(* IEC 61131-3 sources: NVM-AquaFeed-Platform/02_Software_Design/PLC/07_Implementation/Function_Blocks (part 2) *)

(* ---- FB_LineManager.st ---- *)
FUNCTION_BLOCK FB_LineManager
VAR_INPUT
    xEnableFromSystem : BOOL;
    xStart : BOOL;
    xPause : BOOL;
    xStop : BOOL;
    xCancel : BOOL;
    udiCommandSequence : UDINT;
    udiResetSequence : UDINT;
    xEmergencyStop : BOOL;
    xSafetyOK : BOOL;
    xBlockingFault : BOOL;
    xDesktopCommunicationOK : BOOL;
    stConfig : ST_LineConfig;
    udiMonotonicTickMs : UDINT;

    xJobAvailable : BOOL;
    xAcceptJob : BOOL;
    xCandidateIntegrityValid : BOOL;
    stJobCandidate : ST_JobExecution;
    stRecipeCandidate : ST_RecipeExecution;

    xSelectorReady : BOOL;
    xSelectorInPosition : BOOL;
    uiSelectorOutlet : UINT;
    xSelectorFault : BOOL;

    xBlowerReady : BOOL;
    xBlowerRunning : BOOL;
    xBlowerAtSpeed : BOOL;
    xBlowerDosingPermitted : BOOL;
    xBlowerFault : BOOL;

    xDosing1Ready : BOOL;
    xDosing1Running : BOOL;
    xDosing1Fault : BOOL;
    xDosing1CompletedEvent : BOOL;
    udiDosing1DeliveredCentiKg : UDINT;
    udiDosing1IncrementCentiKg : UDINT;

    xDosing2Ready : BOOL;
    xDosing2Running : BOOL;
    xDosing2Fault : BOOL;
    xDosing2CompletedEvent : BOOL;
    udiDosing2DeliveredCentiKg : UDINT;
    udiDosing2IncrementCentiKg : UDINT;
END_VAR
VAR_OUTPUT
    stLine : ST_Line;
    xReady : BOOL;
    xBusy : BOOL;
    xCompleted : BOOL;
    xJobAccepted : BOOL;
    xJobRejected : BOOL;
    uiResultCode : UINT;
    udiLastAcceptedCommandSequence : UDINT;

    xSelectorMoveRequest : BOOL;
    uiSelectorTargetOutlet : UINT;
    udiSelectorCommandSequence : UDINT;

    xBlowerRunRequest : BOOL;
    xBlowerNormalStopRequest : BOOL;
    uiBlowerTargetFreqCentiHz : UINT;
    udiBlowerRequestedPostRunTimeMs : UDINT;
    udiBlowerCommandSequence : UDINT;

    xDosing1StartRequest : BOOL;
    xDosing1StopRequest : BOOL;
    udiDosing1CommandSequence : UDINT;
    udiDosing1JobId : UDINT;
    uiDosing1OutletId : UINT;
    udiDosing1TargetCentiKg : UDINT;
    uiDosing1SpeedPermille : UINT;

    xDosing2StartRequest : BOOL;
    xDosing2StopRequest : BOOL;
    udiDosing2CommandSequence : UDINT;
    udiDosing2JobId : UDINT;
    uiDosing2OutletId : UINT;
    udiDosing2TargetCentiKg : UDINT;
    uiDosing2SpeedPermille : UINT;

    xEquipmentResetRequest : BOOL;
    udiEquipmentResetSequence : UDINT;
END_VAR
VAR
    eState : E_LineState := LINE_OFF;
    stAcceptedJob : ST_JobExecution;
    stAcceptedRecipe : ST_RecipeExecution;
    xActiveJobValid : BOOL;
    xConfigValid : BOOL;
    xCandidateValid : BOOL;
    xSelectedDosingReady : BOOL;
    xSelectedDosingRunning : BOOL;
    xSelectedDosingFault : BOOL;
    xSelectedDosingComplete : BOOL;
    udiSelectedDosingIncrement : UDINT;
    udiSelectedDosingTarget : UDINT;
    udiExecutionStartTickMs : UDINT;
    udiStateStartTickMs : UDINT;
    udiLastResetSequence : UDINT;
    udiLastProcessedTransferSequence : UDINT;
    udiInternalCommandSequence : UDINT;
    xHasAcceptedCommand : BOOL;
    xHasAcceptedReset : BOOL;
    xHasProcessedTransfer : BOOL;
    xShutdownForPause : BOOL;
    xShutdownForCancel : BOOL;
    xShutdownForStop : BOOL;
    xSelectorSettleTimerActive : BOOL;
    xCompleteEventIssued : BOOL;
END_VAR
VAR CONSTANT
    c_udiMaximumProgressTarget : UDINT := 4000000;
    c_udiMaximumExecutionTimeSec : UDINT := 4294967;
    c_uiResultNone : UINT := 0;
    c_uiResultAccepted : UINT := 1;
    c_uiResultCompleted : UINT := 2;
    c_uiResultStopped : UINT := 3;
    c_uiResultCancelled : UINT := 4;
    c_uiResultInvalidConfig : UINT := 60;
    c_uiResultDesktopOffline : UINT := 61;
    c_uiResultIntegrity : UINT := 62;
    c_uiResultInvalidCandidate : UINT := 63;
    c_uiResultEquipmentNotReady : UINT := 64;
    c_uiResultEquipmentFault : UINT := 65;
    c_uiResultSafety : UINT := 66;
    c_uiResultEmergency : UINT := 67;
    c_uiResultTimeout : UINT := 68;
    c_uiResultSequenceOverflow : UINT := 69;
    c_uiResultArithmetic : UINT := 70;
END_VAR

xReady := FALSE;
xBusy := xActiveJobValid;
xCompleted := FALSE;
xJobAccepted := FALSE;
xJobRejected := FALSE;
xSelectorMoveRequest := FALSE;
uiSelectorTargetOutlet := 0;
xBlowerRunRequest := FALSE;
xBlowerNormalStopRequest := FALSE;
uiBlowerTargetFreqCentiHz := 0;
udiBlowerRequestedPostRunTimeMs := 0;
xDosing1StartRequest := FALSE;
xDosing1StopRequest := FALSE;
udiDosing1JobId := 0;
uiDosing1OutletId := 0;
udiDosing1TargetCentiKg := 0;
uiDosing1SpeedPermille := 0;
xDosing2StartRequest := FALSE;
xDosing2StopRequest := FALSE;
udiDosing2JobId := 0;
uiDosing2OutletId := 0;
udiDosing2TargetCentiKg := 0;
uiDosing2SpeedPermille := 0;
xEquipmentResetRequest := FALSE;

xConfigValid := (stConfig.usiLineId > 0) AND
                (stConfig.uiSelectorOutletCount > 0) AND
                (stConfig.uiSelectorOutletCount <= 64) AND
                (stConfig.xDosing1Enabled OR
                 stConfig.xDosing2Enabled) AND
                (stConfig.udiMaximumTargetCentiKg > 0) AND
                (stConfig.udiMaximumTargetCentiKg <=
                 c_udiMaximumProgressTarget) AND
                (stConfig.udiMaximumFeedToleranceCentiKg <
                 stConfig.udiMaximumTargetCentiKg) AND
                (stConfig.uiMinimumDosingSpeedPermille > 0) AND
                (stConfig.uiMinimumDosingSpeedPermille <=
                 stConfig.uiMaximumDosingSpeedPermille) AND
                (stConfig.uiMaximumDosingSpeedPermille <= 1000) AND
                (stConfig.uiMinimumBlowerFreqCentiHz > 0) AND
                (stConfig.uiMinimumBlowerFreqCentiHz <=
                 stConfig.uiMaximumBlowerFreqCentiHz) AND
                (stConfig.udiMaximumSelectorSettleTimeMs > 0) AND
                (stConfig.udiMaximumBlowerPreRunTimeMs > 0) AND
                (stConfig.udiMaximumBlowerPostRunTimeMs > 0) AND
                (stConfig.udiMaximumDosingTimeSec > 0) AND
                (stConfig.udiMaximumExecutionTimeSec > 0) AND
                (stConfig.udiMaximumExecutionTimeSec <=
                 c_udiMaximumExecutionTimeSec);

xCandidateValid := xJobAvailable AND
                   xCandidateIntegrityValid AND
                   (stJobCandidate.uiSnapshotVersion = 1) AND
                   (stRecipeCandidate.uiSnapshotVersion = 1) AND
                   (stJobCandidate.udiJobId > 0) AND
                   (stJobCandidate.usiLineId =
                    stConfig.usiLineId) AND
                   (stJobCandidate.uiRecipeId > 0) AND
                   (stJobCandidate.uiRecipeId =
                    stRecipeCandidate.uiRecipeId) AND
                   (stJobCandidate.udiRecipeRevision =
                    stRecipeCandidate.udiRecipeRevision) AND
                   (stJobCandidate.uiTargetSelectorOutlet > 0) AND
                   (stJobCandidate.uiTargetSelectorOutlet <=
                    stConfig.uiSelectorOutletCount) AND
                   (((stJobCandidate.byDosingUnitMask = 16#01) AND
                     stConfig.xDosing1Enabled) OR
                    ((stJobCandidate.byDosingUnitMask = 16#02) AND
                     stConfig.xDosing2Enabled)) AND
                   (stJobCandidate.udiTargetFeedCentiKg > 0) AND
                   (stJobCandidate.udiTargetFeedCentiKg <=
                    stConfig.udiMaximumTargetCentiKg) AND
                   (stRecipeCandidate.udiFeedToleranceCentiKg <=
                    stConfig.udiMaximumFeedToleranceCentiKg) AND
                   (stRecipeCandidate.udiFeedToleranceCentiKg <
                    stJobCandidate.udiTargetFeedCentiKg) AND
                   (stRecipeCandidate.uiDosingSpeedPermille >=
                    stConfig.uiMinimumDosingSpeedPermille) AND
                   (stRecipeCandidate.uiDosingSpeedPermille <=
                    stConfig.uiMaximumDosingSpeedPermille) AND
                   (stRecipeCandidate.uiBlowerFreqCentiHz >=
                    stConfig.uiMinimumBlowerFreqCentiHz) AND
                   (stRecipeCandidate.uiBlowerFreqCentiHz <=
                    stConfig.uiMaximumBlowerFreqCentiHz) AND
                   (stRecipeCandidate.udiSelectorSettleTimeMs <=
                    stConfig.udiMaximumSelectorSettleTimeMs) AND
                   (stRecipeCandidate.udiBlowerPreRunTimeMs <=
                    stConfig.udiMaximumBlowerPreRunTimeMs) AND
                   (stRecipeCandidate.udiBlowerPostRunTimeMs > 0) AND
                   (stRecipeCandidate.udiBlowerPostRunTimeMs <=
                    stConfig.udiMaximumBlowerPostRunTimeMs) AND
                   (stRecipeCandidate.udiMaximumDosingTimeSec > 0) AND
                   (stRecipeCandidate.udiMaximumDosingTimeSec <=
                    stConfig.udiMaximumDosingTimeSec) AND
                   (stJobCandidate.udiMaximumExecutionTimeSec > 0) AND
                   (stJobCandidate.udiMaximumExecutionTimeSec <=
                    stConfig.udiMaximumExecutionTimeSec);

xSelectedDosingReady := FALSE;
xSelectedDosingRunning := FALSE;
xSelectedDosingFault := FALSE;
xSelectedDosingComplete := FALSE;
udiSelectedDosingIncrement := 0;

IF xActiveJobValid THEN
    IF stAcceptedJob.byDosingUnitMask = 16#01 THEN
        xSelectedDosingReady := xDosing1Ready;
        xSelectedDosingRunning := xDosing1Running;
        xSelectedDosingFault := xDosing1Fault;
        xSelectedDosingComplete := xDosing1CompletedEvent;
        udiSelectedDosingIncrement :=
            udiDosing1IncrementCentiKg;
    ELSIF stAcceptedJob.byDosingUnitMask = 16#02 THEN
        xSelectedDosingReady := xDosing2Ready;
        xSelectedDosingRunning := xDosing2Running;
        xSelectedDosingFault := xDosing2Fault;
        xSelectedDosingComplete := xDosing2CompletedEvent;
        udiSelectedDosingIncrement :=
            udiDosing2IncrementCentiKg;
    END_IF;
END_IF;

IF NOT xEnableFromSystem THEN
    eState := LINE_OFF;
    xActiveJobValid := FALSE;
    xShutdownForPause := FALSE;
    xShutdownForCancel := FALSE;
    xShutdownForStop := FALSE;
    xCompleteEventIssued := FALSE;
    uiResultCode := c_uiResultNone;
ELSIF NOT xConfigValid THEN
    eState := LINE_FAULT;
    uiResultCode := c_uiResultInvalidConfig;
ELSIF xEmergencyStop THEN
    eState := LINE_EMERGENCY;
    uiResultCode := c_uiResultEmergency;
ELSIF xActiveJobValid AND
      (NOT xSafetyOK OR xBlockingFault) THEN
    eState := LINE_FAULT;
    uiResultCode := c_uiResultSafety;
ELSIF xActiveJobValid AND
      (xSelectorFault OR xBlowerFault OR
       xSelectedDosingFault) THEN
    eState := LINE_FAULT;
    uiResultCode := c_uiResultEquipmentFault;
ELSE
    IF xActiveJobValid AND
       (eState <> LINE_PAUSED) AND
       (eState <> LINE_FAULT) AND
       (eState <> LINE_EMERGENCY) AND
       (F_ElapsedMs(udiCurrentTickMs := udiMonotonicTickMs,
                    udiStartTickMs := udiExecutionStartTickMs) >=
        (stAcceptedJob.udiMaximumExecutionTimeSec * 1000)) THEN
        eState := LINE_FAULT;
        uiResultCode := c_uiResultTimeout;
    END_IF;

    IF xActiveJobValid AND
       (eState <> LINE_LOAD_JOB) AND
       (eState <> LINE_READY) AND
       (eState <> LINE_PAUSED) AND
       (eState <> LINE_FAULT) AND
       (eState <> LINE_EMERGENCY) AND
       (NOT xHasAcceptedCommand OR
        (udiCommandSequence <>
         udiLastAcceptedCommandSequence)) THEN
        IF xCancel OR xStop OR xPause THEN
            udiLastAcceptedCommandSequence :=
                udiCommandSequence;
            xHasAcceptedCommand := TRUE;
            xShutdownForCancel := xCancel;
            xShutdownForStop := xStop AND NOT xCancel;
            xShutdownForPause :=
                xPause AND NOT xStop AND NOT xCancel;
            eState := LINE_STOP_DOSING;
        END_IF;
    END_IF;

    CASE eState OF
        LINE_OFF:
            eState := LINE_INITIALIZING;
            uiResultCode := c_uiResultNone;

        LINE_INITIALIZING:
            IF xSafetyOK AND
               NOT xBlockingFault AND
               NOT xSelectorFault AND
               NOT xBlowerFault THEN
                eState := LINE_READY;
            END_IF;

        LINE_READY:
            xReady := TRUE;

            IF xAcceptJob AND
               (NOT xHasProcessedTransfer OR
                (stJobCandidate.udiTransferSequence <>
                 udiLastProcessedTransferSequence)) THEN
                udiLastProcessedTransferSequence :=
                    stJobCandidate.udiTransferSequence;
                xHasProcessedTransfer := TRUE;

                IF NOT xDesktopCommunicationOK THEN
                    xJobRejected := TRUE;
                    uiResultCode := c_uiResultDesktopOffline;
                ELSIF NOT xCandidateIntegrityValid THEN
                    xJobRejected := TRUE;
                    uiResultCode := c_uiResultIntegrity;
                ELSIF NOT xCandidateValid THEN
                    xJobRejected := TRUE;
                    uiResultCode := c_uiResultInvalidCandidate;
                ELSE
                    stAcceptedJob := stJobCandidate;
                    stAcceptedRecipe := stRecipeCandidate;
                    xActiveJobValid := TRUE;
                    xJobAccepted := TRUE;
                    xShutdownForPause := FALSE;
                    xShutdownForCancel := FALSE;
                    xShutdownForStop := FALSE;
                    xCompleteEventIssued := FALSE;
                    stLine.udiDeliveredFeedCentiKg := 0;
                    uiResultCode := c_uiResultAccepted;
                    eState := LINE_LOAD_JOB;
                END_IF;
            END_IF;

        LINE_LOAD_JOB:
            IF xStart AND
               (NOT xHasAcceptedCommand OR
                (udiCommandSequence <>
                 udiLastAcceptedCommandSequence)) THEN
                udiLastAcceptedCommandSequence :=
                    udiCommandSequence;
                xHasAcceptedCommand := TRUE;
                udiExecutionStartTickMs :=
                    udiMonotonicTickMs;
                eState := LINE_VALIDATE;
            END_IF;

        LINE_VALIDATE:
            IF NOT xSafetyOK OR xBlockingFault OR
               NOT xSelectorReady OR
               NOT xBlowerReady OR
               NOT xSelectedDosingReady THEN
                eState := LINE_FAULT;
                uiResultCode := c_uiResultEquipmentNotReady;
            ELSIF udiInternalCommandSequence =
                  16#FFFFFFFF THEN
                eState := LINE_FAULT;
                uiResultCode := c_uiResultSequenceOverflow;
            ELSE
                udiInternalCommandSequence :=
                    udiInternalCommandSequence + 1;
                udiSelectorCommandSequence :=
                    udiInternalCommandSequence;
                eState := LINE_MOVE_SELECTOR;
            END_IF;

        LINE_MOVE_SELECTOR:
            xSelectorMoveRequest := TRUE;
            uiSelectorTargetOutlet :=
                stAcceptedJob.uiTargetSelectorOutlet;
            eState := LINE_WAIT_SELECTOR;
            xSelectorSettleTimerActive := FALSE;

        LINE_WAIT_SELECTOR:
            uiSelectorTargetOutlet :=
                stAcceptedJob.uiTargetSelectorOutlet;

            IF xSelectorInPosition AND
               (uiSelectorOutlet =
                stAcceptedJob.uiTargetSelectorOutlet) THEN
                IF NOT xSelectorSettleTimerActive THEN
                    udiStateStartTickMs :=
                        udiMonotonicTickMs;
                    xSelectorSettleTimerActive := TRUE;
                ELSIF F_ElapsedMs(
                          udiCurrentTickMs :=
                              udiMonotonicTickMs,
                          udiStartTickMs :=
                              udiStateStartTickMs) >=
                      stAcceptedRecipe.
                          udiSelectorSettleTimeMs THEN
                    eState := LINE_START_BLOWER;
                END_IF;
            ELSE
                xSelectorSettleTimerActive := FALSE;
            END_IF;

        LINE_START_BLOWER:
            IF udiInternalCommandSequence =
               16#FFFFFFFF THEN
                eState := LINE_FAULT;
                uiResultCode := c_uiResultSequenceOverflow;
            ELSE
                udiInternalCommandSequence :=
                    udiInternalCommandSequence + 1;
                udiBlowerCommandSequence :=
                    udiInternalCommandSequence;
                eState := LINE_WAIT_BLOWER;
            END_IF;

        LINE_WAIT_BLOWER:
            xBlowerRunRequest := TRUE;
            uiBlowerTargetFreqCentiHz :=
                stAcceptedRecipe.uiBlowerFreqCentiHz;
            udiBlowerRequestedPostRunTimeMs :=
                stAcceptedRecipe.udiBlowerPostRunTimeMs;

            IF xBlowerAtSpeed AND
               xBlowerDosingPermitted THEN
                udiStateStartTickMs :=
                    udiMonotonicTickMs;
                eState := LINE_PRE_RUN;
            END_IF;

        LINE_PRE_RUN:
            xBlowerRunRequest := TRUE;
            uiBlowerTargetFreqCentiHz :=
                stAcceptedRecipe.uiBlowerFreqCentiHz;
            udiBlowerRequestedPostRunTimeMs :=
                stAcceptedRecipe.udiBlowerPostRunTimeMs;

            IF NOT xSelectorInPosition OR
               (uiSelectorOutlet <>
                stAcceptedJob.uiTargetSelectorOutlet) OR
               NOT xBlowerDosingPermitted THEN
                eState := LINE_FAULT;
                uiResultCode := c_uiResultEquipmentFault;
            ELSIF F_ElapsedMs(
                      udiCurrentTickMs :=
                          udiMonotonicTickMs,
                      udiStartTickMs :=
                          udiStateStartTickMs) >=
                  stAcceptedRecipe.
                      udiBlowerPreRunTimeMs THEN
                eState := LINE_START_DOSING;
            END_IF;

        LINE_START_DOSING:
            xBlowerRunRequest := TRUE;
            uiBlowerTargetFreqCentiHz :=
                stAcceptedRecipe.uiBlowerFreqCentiHz;
            udiBlowerRequestedPostRunTimeMs :=
                stAcceptedRecipe.udiBlowerPostRunTimeMs;

            IF udiInternalCommandSequence =
               16#FFFFFFFF THEN
                eState := LINE_FAULT;
                uiResultCode := c_uiResultSequenceOverflow;
            ELSE
                udiInternalCommandSequence :=
                    udiInternalCommandSequence + 1;
                IF stAcceptedJob.byDosingUnitMask =
                   16#01 THEN
                    udiDosing1CommandSequence :=
                        udiInternalCommandSequence;
                ELSE
                    udiDosing2CommandSequence :=
                        udiInternalCommandSequence;
                END_IF;

                IF stLine.udiDeliveredFeedCentiKg >=
                   stAcceptedJob.udiTargetFeedCentiKg THEN
                    udiSelectedDosingTarget := 0;
                ELSE
                    udiSelectedDosingTarget :=
                        stAcceptedJob.
                            udiTargetFeedCentiKg -
                        stLine.
                            udiDeliveredFeedCentiKg;
                END_IF;
                eState := LINE_FEEDING;
            END_IF;

        LINE_FEEDING:
            xBlowerRunRequest := TRUE;
            uiBlowerTargetFreqCentiHz :=
                stAcceptedRecipe.uiBlowerFreqCentiHz;
            udiBlowerRequestedPostRunTimeMs :=
                stAcceptedRecipe.udiBlowerPostRunTimeMs;

            IF stAcceptedJob.byDosingUnitMask = 16#01 THEN
                xDosing1StartRequest := TRUE;
                udiDosing1JobId := stAcceptedJob.udiJobId;
                uiDosing1OutletId :=
                    stAcceptedJob.uiTargetSelectorOutlet;
                udiDosing1TargetCentiKg :=
                    udiSelectedDosingTarget;
                uiDosing1SpeedPermille :=
                    stAcceptedRecipe.uiDosingSpeedPermille;
            ELSE
                xDosing2StartRequest := TRUE;
                udiDosing2JobId := stAcceptedJob.udiJobId;
                uiDosing2OutletId :=
                    stAcceptedJob.uiTargetSelectorOutlet;
                udiDosing2TargetCentiKg :=
                    udiSelectedDosingTarget;
                uiDosing2SpeedPermille :=
                    stAcceptedRecipe.uiDosingSpeedPermille;
            END_IF;

            IF NOT xSelectorInPosition OR
               (uiSelectorOutlet <>
                stAcceptedJob.uiTargetSelectorOutlet) OR
               NOT xBlowerDosingPermitted THEN
                eState := LINE_FAULT;
                uiResultCode := c_uiResultEquipmentFault;
            ELSE
                IF stLine.udiDeliveredFeedCentiKg >=
                   stAcceptedJob.udiTargetFeedCentiKg THEN
                    stLine.udiDeliveredFeedCentiKg :=
                        stAcceptedJob.udiTargetFeedCentiKg;
                ELSIF udiSelectedDosingIncrement >=
                      (stAcceptedJob.udiTargetFeedCentiKg -
                       stLine.udiDeliveredFeedCentiKg) THEN
                    stLine.udiDeliveredFeedCentiKg :=
                        stAcceptedJob.udiTargetFeedCentiKg;
                ELSE
                    stLine.udiDeliveredFeedCentiKg :=
                        stLine.udiDeliveredFeedCentiKg +
                        udiSelectedDosingIncrement;
                END_IF;

                IF xSelectedDosingComplete THEN
                    eState := LINE_STOP_DOSING;
                END_IF;
            END_IF;

        LINE_STOP_DOSING:
            xBlowerRunRequest := xBlowerRunning;
            uiBlowerTargetFreqCentiHz :=
                stAcceptedRecipe.uiBlowerFreqCentiHz;
            udiBlowerRequestedPostRunTimeMs :=
                stAcceptedRecipe.udiBlowerPostRunTimeMs;

            IF stAcceptedJob.byDosingUnitMask = 16#01 THEN
                xDosing1StopRequest := TRUE;
            ELSE
                xDosing2StopRequest := TRUE;
            END_IF;

            IF NOT xSelectedDosingRunning THEN
                eState := LINE_POST_RUN;
            END_IF;

        LINE_POST_RUN:
            xBlowerRunRequest := TRUE;
            xBlowerNormalStopRequest := TRUE;
            uiBlowerTargetFreqCentiHz :=
                stAcceptedRecipe.uiBlowerFreqCentiHz;
            udiBlowerRequestedPostRunTimeMs :=
                stAcceptedRecipe.udiBlowerPostRunTimeMs;

            IF NOT xBlowerRunning AND xBlowerReady THEN
                IF xShutdownForPause THEN
                    eState := LINE_PAUSED;
                ELSIF xShutdownForCancel THEN
                    xActiveJobValid := FALSE;
                    uiResultCode := c_uiResultCancelled;
                    eState := LINE_READY;
                ELSIF xShutdownForStop THEN
                    xActiveJobValid := FALSE;
                    uiResultCode := c_uiResultStopped;
                    eState := LINE_READY;
                ELSE
                    eState := LINE_COMPLETE;
                    xCompleteEventIssued := FALSE;
                END_IF;
            END_IF;

        LINE_COMPLETE:
            IF NOT xCompleteEventIssued THEN
                xCompleted := TRUE;
                xCompleteEventIssued := TRUE;
                uiResultCode := c_uiResultCompleted;
            ELSE
                xActiveJobValid := FALSE;
                xCompleteEventIssued := FALSE;
                eState := LINE_READY;
            END_IF;

        LINE_PAUSED:
            IF xStart AND
               (NOT xHasAcceptedCommand OR
                (udiCommandSequence <>
                 udiLastAcceptedCommandSequence)) AND
               xSafetyOK AND
               NOT xBlockingFault THEN
                udiLastAcceptedCommandSequence :=
                    udiCommandSequence;
                xHasAcceptedCommand := TRUE;
                xShutdownForPause := FALSE;
                xShutdownForCancel := FALSE;
                xShutdownForStop := FALSE;
                eState := LINE_VALIDATE;
            ELSIF (xCancel OR xStop) AND
                  (NOT xHasAcceptedCommand OR
                   (udiCommandSequence <>
                    udiLastAcceptedCommandSequence)) THEN
                udiLastAcceptedCommandSequence :=
                    udiCommandSequence;
                xHasAcceptedCommand := TRUE;
                xActiveJobValid := FALSE;
                IF xCancel THEN
                    uiResultCode := c_uiResultCancelled;
                ELSE
                    uiResultCode := c_uiResultStopped;
                END_IF;
                eState := LINE_READY;
            END_IF;

        LINE_STOPPING:
            eState := LINE_STOP_DOSING;

        LINE_RECOVERY:
            eState := LINE_VALIDATE;

        LINE_FAULT:
            IF (NOT xHasAcceptedReset OR
                (udiResetSequence <> udiLastResetSequence)) AND
               NOT xEmergencyStop AND
               xSafetyOK AND
               NOT xBlockingFault AND
               NOT xSelectorFault AND
               NOT xBlowerFault AND
               NOT xSelectedDosingFault AND
               NOT xSelectorMoveRequest AND
               NOT xBlowerRunning AND
               NOT xSelectedDosingRunning THEN
                udiLastResetSequence := udiResetSequence;
                xHasAcceptedReset := TRUE;
                udiEquipmentResetSequence :=
                    udiResetSequence;
                xEquipmentResetRequest := TRUE;
                xActiveJobValid := FALSE;
                xShutdownForPause := FALSE;
                xShutdownForCancel := FALSE;
                xShutdownForStop := FALSE;
                eState := LINE_INITIALIZING;
                uiResultCode := c_uiResultNone;
            END_IF;

        LINE_EMERGENCY:
            IF (NOT xHasAcceptedReset OR
                (udiResetSequence <> udiLastResetSequence)) AND
               NOT xEmergencyStop AND
               xSafetyOK AND
               NOT xBlockingFault AND
               NOT xBlowerRunning AND
               NOT xSelectedDosingRunning THEN
                udiLastResetSequence := udiResetSequence;
                xHasAcceptedReset := TRUE;
                udiEquipmentResetSequence :=
                    udiResetSequence;
                xEquipmentResetRequest := TRUE;
                xActiveJobValid := FALSE;
                eState := LINE_INITIALIZING;
                uiResultCode := c_uiResultNone;
            END_IF;

        LINE_SERVICE:
            eState := LINE_READY;

    ELSE
        eState := LINE_FAULT;
        uiResultCode := c_uiResultInvalidConfig;
    END_CASE;
END_IF;

IF (eState = LINE_FAULT) OR
   (eState = LINE_EMERGENCY) OR
   (eState = LINE_OFF) THEN
    xSelectorMoveRequest := FALSE;
    xBlowerRunRequest := FALSE;
    xBlowerNormalStopRequest := FALSE;
    xDosing1StartRequest := FALSE;
    xDosing2StartRequest := FALSE;
END_IF;

IF xActiveJobValid THEN
    IF stLine.udiDeliveredFeedCentiKg >=
       stAcceptedJob.udiTargetFeedCentiKg THEN
        stLine.udiRemainingFeedCentiKg := 0;
        stLine.uiProgressPermille := 1000;
    ELSE
        stLine.udiRemainingFeedCentiKg :=
            stAcceptedJob.udiTargetFeedCentiKg -
            stLine.udiDeliveredFeedCentiKg;
        stLine.uiProgressPermille :=
            UDINT_TO_UINT(
                (stLine.udiDeliveredFeedCentiKg * 1000) /
                stAcceptedJob.udiTargetFeedCentiKg);
    END_IF;
ELSE
    stLine.udiRemainingFeedCentiKg := 0;
    stLine.uiProgressPermille := 0;
END_IF;

stLine.usiLineId := stConfig.usiLineId;
stLine.eLineState := eState;
stLine.xEnabled := xEnableFromSystem;
stLine.xReady := xReady;
stLine.xBusy := xActiveJobValid;
stLine.xRunning := (eState >= LINE_MOVE_SELECTOR) AND
                   (eState <= LINE_POST_RUN);
stLine.xPaused := eState = LINE_PAUSED;
stLine.xCompleted := xCompleted;
stLine.xFault := eState = LINE_FAULT;
stLine.xEmergency := eState = LINE_EMERGENCY;
stLine.xAutoMode := TRUE;
stLine.xManualMode := FALSE;
stLine.xServiceMode := FALSE;
stLine.xSimulationMode := FALSE;
stLine.xActiveJobValid := xActiveJobValid;
stLine.uiCurrentSelectorOutlet := uiSelectorOutlet;
stLine.udiRemainingTimeSec := 0;

IF xActiveJobValid THEN
    stLine.udiActiveJobId := stAcceptedJob.udiJobId;
    stLine.uiActiveRecipeId := stAcceptedJob.uiRecipeId;
    stLine.uiTargetSelectorOutlet :=
        stAcceptedJob.uiTargetSelectorOutlet;
    stLine.xSelectorAtTarget :=
        xSelectorInPosition AND
        (uiSelectorOutlet =
         stAcceptedJob.uiTargetSelectorOutlet);
    stLine.udiTargetFeedCentiKg :=
        stAcceptedJob.udiTargetFeedCentiKg;
    stLine.udiElapsedTimeSec :=
        F_ElapsedMs(udiCurrentTickMs := udiMonotonicTickMs,
                    udiStartTickMs := udiExecutionStartTickMs) /
        1000;
ELSE
    stLine.udiActiveJobId := 0;
    stLine.uiActiveRecipeId := 0;
    stLine.uiTargetSelectorOutlet := 0;
    stLine.xSelectorAtTarget := FALSE;
    stLine.udiTargetFeedCentiKg := 0;
    stLine.udiDeliveredFeedCentiKg := 0;
    stLine.udiElapsedTimeSec := 0;
END_IF;
stLine.xBlowerRunning := xBlowerRunning;
stLine.xDosing1Running := xDosing1Running;
stLine.xDosing2Running := xDosing2Running;
stLine.uiActiveAlarmId := 0;

xReady := eState = LINE_READY;
xBusy := xActiveJobValid;

END_FUNCTION_BLOCK

(* ---- FB_RecoveryManager.st ---- *)
FUNCTION_BLOCK FB_RecoveryManager
VAR_INPUT
    xEvaluateRequest : BOOL;
    xResumeApproval : BOOL;
    xRejectRequest : BOOL;
    udiRecoverySequence : UDINT;
    xCheckpointPresent : BOOL;
    stCheckpoint : ST_RecoveryCheckpoint;
    xCheckpointIntegrityValid : BOOL;
    xDesktopCheckpointStillCurrent : BOOL;
    xSafetyRecoveryPermitted : BOOL;
    xEquipmentStopped : BOOL;
    xEquipmentFeedbackKnown : BOOL;
    xConfigurationValid : BOOL;
    xIOHealthy : BOOL;
    xCommunicationHealthy : BOOL;
    xSelectorReady : BOOL;
    xBlowerReady : BOOL;
    xDosingReady : BOOL;
    xReinitializationComplete : BOOL;
    xReinitializationFailed : BOOL;
    xLineResumeAccepted : BOOL;
END_VAR
VAR_OUTPUT
    stRecovery : ST_RecoveryStatus;
    stApprovedJob : ST_JobExecution;
    stApprovedRecipe : ST_RecipeExecution;
    udiApprovedDeliveredCentiKg : UDINT;
    xReinitializeRequest : BOOL;
    xResumeCommandAccepted : BOOL;
    xRequestRejected : BOOL;
END_VAR
VAR
    stAcceptedCheckpoint : ST_RecoveryCheckpoint;
    xHasProcessedRequest : BOOL;
    udiLastProcessedSequence : UDINT;
    xCommandConflict : BOOL;
    xNewRequest : BOOL;
    xLiveValid : BOOL;
    xSnapshotValid : BOOL;
END_VAR
VAR CONSTANT
    c_uiResultNone : UINT := 0;
    c_uiResultCommandConflict : UINT := 1;
    c_uiResultCheckpointMissing : UINT := 10;
    c_uiResultIntegrityInvalid : UINT := 11;
    c_uiResultSnapshotInvalid : UINT := 12;
    c_uiResultQuantityInvalid : UINT := 13;
    c_uiResultTerminalExecution : UINT := 14;
    c_uiResultRetryExhausted : UINT := 15;
    c_uiResultDesktopSuperseded : UINT := 20;
    c_uiResultSafetyBlocked : UINT := 21;
    c_uiResultEquipmentUnknown : UINT := 22;
    c_uiResultPrerequisiteFailed : UINT := 23;
    c_uiResultReinitializationFailed : UINT := 30;
    c_uiResultSequenceExhausted : UINT := 31;
    c_uiResultUnknownState : UINT := 90;
END_VAR

xReinitializeRequest := FALSE;
xResumeCommandAccepted := FALSE;
xRequestRejected := FALSE;
stRecovery.xRecoveryAvailable := FALSE;
stRecovery.xApprovalRequired := FALSE;
stRecovery.xReadyToResume := FALSE;
stRecovery.xApprovedCheckpointValid := FALSE;

xCommandConflict := (xEvaluateRequest AND xResumeApproval) OR
                    (xEvaluateRequest AND xRejectRequest) OR
                    (xResumeApproval AND xRejectRequest);
xNewRequest := (xEvaluateRequest OR xResumeApproval OR xRejectRequest) AND
               (NOT xHasProcessedRequest OR
                (udiRecoverySequence <> udiLastProcessedSequence));

xLiveValid := xDesktopCheckpointStillCurrent AND
              xSafetyRecoveryPermitted AND
              xEquipmentStopped AND
              xEquipmentFeedbackKnown AND
              xConfigurationValid AND
              xIOHealthy AND
              xCommunicationHealthy AND
              xSelectorReady AND
              xBlowerReady AND
              xDosingReady;

IF xNewRequest THEN
    IF xHasProcessedRequest AND
       (udiLastProcessedSequence = 16#FFFFFFFF) AND
       (udiRecoverySequence = 0) THEN
        stRecovery.eState := RecoveryFailed;
        stRecovery.uiResultCode := c_uiResultSequenceExhausted;
        xRequestRejected := TRUE;
    ELSE
        xHasProcessedRequest := TRUE;
        udiLastProcessedSequence := udiRecoverySequence;
        stRecovery.udiLastProcessedRecoverySequence := udiRecoverySequence;

        IF xCommandConflict THEN
            xRequestRejected := TRUE;
            stRecovery.uiResultCode := c_uiResultCommandConflict;
        ELSIF xRejectRequest THEN
            stRecovery.eState := RecoveryRejected;
            stRecovery.uiResultCode := c_uiResultNone;
            xRequestRejected := TRUE;
        ELSIF xEvaluateRequest THEN
            stAcceptedCheckpoint := stCheckpoint;
            stRecovery.eState := RecoveryEvaluating;
            stRecovery.uiResultCode := c_uiResultNone;
        ELSIF xResumeApproval THEN
            IF stRecovery.eState <> RecoveryAwaitingApproval THEN
                xRequestRejected := TRUE;
                stRecovery.uiResultCode := c_uiResultSnapshotInvalid;
            ELSIF NOT xLiveValid THEN
                xRequestRejected := TRUE;
                stRecovery.eState := RecoveryFailed;
                stRecovery.uiResultCode := c_uiResultPrerequisiteFailed;
            ELSE
                stRecovery.eState := RecoveryReinitializing;
                stRecovery.uiResultCode := c_uiResultNone;
                xResumeCommandAccepted := TRUE;
            END_IF;
        END_IF;
    END_IF;
END_IF;

CASE stRecovery.eState OF
    RecoveryIdle:
        stRecovery.uiResultCode := c_uiResultNone;

    RecoveryEvaluating:
        xSnapshotValid :=
            xCheckpointPresent AND
            xCheckpointIntegrityValid AND
            (stAcceptedCheckpoint.uiCheckpointVersion = 1) AND
            (stAcceptedCheckpoint.stJob.uiSnapshotVersion = 1) AND
            (stAcceptedCheckpoint.stRecipe.uiSnapshotVersion = 1) AND
            (stAcceptedCheckpoint.stJob.udiJobId <> 0) AND
            (stAcceptedCheckpoint.stJob.usiLineId <> 0) AND
            (stAcceptedCheckpoint.stJob.uiRecipeId =
             stAcceptedCheckpoint.stRecipe.uiRecipeId) AND
            (stAcceptedCheckpoint.stJob.udiRecipeRevision =
             stAcceptedCheckpoint.stRecipe.udiRecipeRevision) AND
            (stAcceptedCheckpoint.stJob.udiTargetFeedCentiKg > 0) AND
            (stAcceptedCheckpoint.stJob.uiTargetSelectorOutlet > 0) AND
            stAcceptedCheckpoint.stJob.xAllowRecovery;

        stRecovery.xSnapshotPresent := xCheckpointPresent;
        stRecovery.xSnapshotValid := FALSE;

        IF NOT xCheckpointPresent THEN
            stRecovery.eState := RecoveryRejected;
            stRecovery.uiResultCode := c_uiResultCheckpointMissing;
        ELSIF NOT xCheckpointIntegrityValid THEN
            stRecovery.eState := RecoveryRejected;
            stRecovery.uiResultCode := c_uiResultIntegrityInvalid;
        ELSIF NOT xSnapshotValid THEN
            stRecovery.eState := RecoveryRejected;
            stRecovery.uiResultCode := c_uiResultSnapshotInvalid;
        ELSIF stAcceptedCheckpoint.xExecutionCompleted OR
              stAcceptedCheckpoint.xExecutionCancelled THEN
            stRecovery.eState := RecoveryRejected;
            stRecovery.uiResultCode := c_uiResultTerminalExecution;
        ELSIF NOT stAcceptedCheckpoint.xQuantityTrustworthy OR
              (stAcceptedCheckpoint.udiDeliveredFeedCentiKg >
               stAcceptedCheckpoint.stJob.udiTargetFeedCentiKg) THEN
            stRecovery.eState := RecoveryRejected;
            stRecovery.uiResultCode := c_uiResultQuantityInvalid;
        ELSIF stAcceptedCheckpoint.usiRetryCount >=
              stAcceptedCheckpoint.stJob.usiMaximumRetryCount THEN
            stRecovery.eState := RecoveryRejected;
            stRecovery.uiResultCode := c_uiResultRetryExhausted;
        ELSIF NOT xDesktopCheckpointStillCurrent THEN
            stRecovery.eState := RecoveryRejected;
            stRecovery.uiResultCode := c_uiResultDesktopSuperseded;
        ELSIF NOT xSafetyRecoveryPermitted THEN
            stRecovery.eState := RecoveryRejected;
            stRecovery.uiResultCode := c_uiResultSafetyBlocked;
        ELSIF NOT xEquipmentStopped OR NOT xEquipmentFeedbackKnown THEN
            stRecovery.eState := RecoveryRejected;
            stRecovery.uiResultCode := c_uiResultEquipmentUnknown;
        ELSIF NOT xLiveValid THEN
            stRecovery.eState := RecoveryRejected;
            stRecovery.uiResultCode := c_uiResultPrerequisiteFailed;
        ELSE
            stRecovery.xSnapshotValid := TRUE;
            stRecovery.udiJobId := stAcceptedCheckpoint.stJob.udiJobId;
            stRecovery.udiRecipeRevision :=
                stAcceptedCheckpoint.stRecipe.udiRecipeRevision;
            stRecovery.usiLineId := stAcceptedCheckpoint.stJob.usiLineId;
            stRecovery.uiOutletId :=
                stAcceptedCheckpoint.stJob.uiTargetSelectorOutlet;
            stRecovery.udiTargetFeedCentiKg :=
                stAcceptedCheckpoint.stJob.udiTargetFeedCentiKg;
            stRecovery.udiDeliveredCentiKg :=
                stAcceptedCheckpoint.udiDeliveredFeedCentiKg;
            stRecovery.udiRemainingFeedCentiKg :=
                stAcceptedCheckpoint.stJob.udiTargetFeedCentiKg -
                stAcceptedCheckpoint.udiDeliveredFeedCentiKg;
            stRecovery.usiRetryCount := stAcceptedCheckpoint.usiRetryCount;
            stRecovery.udiLastAcceptedCommandSequence :=
                stAcceptedCheckpoint.udiLastAcceptedCommandSequence;
            stRecovery.uiInterruptionReason :=
                stAcceptedCheckpoint.uiInterruptionReason;
            stRecovery.eState := RecoveryAvailable;
            stRecovery.uiResultCode := c_uiResultNone;
        END_IF;

    RecoveryAvailable:
        stRecovery.xRecoveryAvailable := TRUE;
        stRecovery.eState := RecoveryAwaitingApproval;

    RecoveryAwaitingApproval:
        stRecovery.xRecoveryAvailable := TRUE;
        stRecovery.xApprovalRequired := TRUE;

    RecoveryReinitializing:
        IF NOT xLiveValid THEN
            stRecovery.eState := RecoveryFailed;
            stRecovery.uiResultCode := c_uiResultPrerequisiteFailed;
        ELSIF xReinitializationFailed THEN
            stRecovery.eState := RecoveryFailed;
            stRecovery.uiResultCode := c_uiResultReinitializationFailed;
        ELSIF xReinitializationComplete THEN
            stApprovedJob := stAcceptedCheckpoint.stJob;
            stApprovedRecipe := stAcceptedCheckpoint.stRecipe;
            udiApprovedDeliveredCentiKg :=
                stAcceptedCheckpoint.udiDeliveredFeedCentiKg;
            stRecovery.eState := RecoveryReadyToResume;
            stRecovery.uiResultCode := c_uiResultNone;
        ELSE
            xReinitializeRequest := TRUE;
        END_IF;

    RecoveryReadyToResume:
        IF NOT xLiveValid THEN
            stRecovery.eState := RecoveryFailed;
            stRecovery.uiResultCode := c_uiResultPrerequisiteFailed;
        ELSE
            stRecovery.xReadyToResume := TRUE;
            stRecovery.xApprovedCheckpointValid := TRUE;
            IF xLineResumeAccepted THEN
                stRecovery.eState := RecoveryCompleted;
            END_IF;
        END_IF;

    RecoveryCompleted:
        stRecovery.uiResultCode := c_uiResultNone;

    RecoveryRejected:
        stRecovery.xSnapshotValid := FALSE;

    RecoveryFailed:
        stRecovery.xSnapshotValid := FALSE;

ELSE
    stRecovery.eState := RecoveryFailed;
    stRecovery.uiResultCode := c_uiResultUnknownState;
END_CASE;

END_FUNCTION_BLOCK

(* ---- FB_SafetyCoordinator.st ---- *)
FUNCTION_BLOCK FB_SafetyCoordinator
VAR_INPUT
    xFeedbackValid : BOOL;
    xEmergencyActive : BOOL;
    xSafetyRelayHealthy : BOOL;
    xSTOFeedbackHealthy : BOOL;
    xContactorFeedbackHealthy : BOOL;
    xStandardControlPermitRequest : BOOL;

    xLocalResetRequest : BOOL;
    udiResetSequence : UDINT;
    xEquipmentStopped : BOOL;
END_VAR
VAR_OUTPUT
    stSafety : ST_SafetyStatus;
    xResetAccepted : BOOL;
    xResetRejected : BOOL;
END_VAR
VAR
    xResetRequiredLatched : BOOL := TRUE;
    xHasProcessedReset : BOOL;
    udiLastProcessedResetSequence : UDINT;
    xAllObservedHealthy : BOOL;
END_VAR
VAR CONSTANT
    c_uiDiagnosticNone : UINT := 0;
    c_uiDiagnosticFeedbackInvalid : UINT := 50;
    c_uiDiagnosticEmergencyActive : UINT := 51;
    c_uiDiagnosticSafetyRelay : UINT := 52;
    c_uiDiagnosticSTOFeedback : UINT := 53;
    c_uiDiagnosticContactorFeedback : UINT := 54;
    c_uiDiagnosticEquipmentRunning : UINT := 55;
    c_uiDiagnosticPermitRequestActive : UINT := 56;
    c_uiDiagnosticResetNotRequired : UINT := 57;
END_VAR

xResetAccepted := FALSE;
xResetRejected := FALSE;

stSafety.xAutomaticPermitted := FALSE;
stSafety.xMotionPermitted := FALSE;
stSafety.xBlowerPermitted := FALSE;
stSafety.xDosingPermitted := FALSE;
stSafety.xRecoveryPermitted := FALSE;

xAllObservedHealthy := xFeedbackValid AND
                       NOT xEmergencyActive AND
                       xSafetyRelayHealthy AND
                       xSTOFeedbackHealthy AND
                       xContactorFeedbackHealthy;

(* Any unknown, trip, or implausible feedback requires a new local reset. *)
IF NOT xAllObservedHealthy THEN
    xResetRequiredLatched := TRUE;
END_IF;

(* A new sequence is evaluated once; replay produces no result event. *)
IF xLocalResetRequest AND
   (NOT xHasProcessedReset OR
    (udiResetSequence <> udiLastProcessedResetSequence)) THEN
    xHasProcessedReset := TRUE;
    udiLastProcessedResetSequence := udiResetSequence;

    IF NOT xFeedbackValid THEN
        xResetRejected := TRUE;
        stSafety.uiDiagnosticCode :=
            c_uiDiagnosticFeedbackInvalid;
    ELSIF xEmergencyActive THEN
        xResetRejected := TRUE;
        stSafety.uiDiagnosticCode :=
            c_uiDiagnosticEmergencyActive;
    ELSIF NOT xSafetyRelayHealthy THEN
        xResetRejected := TRUE;
        stSafety.uiDiagnosticCode :=
            c_uiDiagnosticSafetyRelay;
    ELSIF NOT xSTOFeedbackHealthy THEN
        xResetRejected := TRUE;
        stSafety.uiDiagnosticCode :=
            c_uiDiagnosticSTOFeedback;
    ELSIF NOT xContactorFeedbackHealthy THEN
        xResetRejected := TRUE;
        stSafety.uiDiagnosticCode :=
            c_uiDiagnosticContactorFeedback;
    ELSIF NOT xResetRequiredLatched THEN
        xResetRejected := TRUE;
        stSafety.uiDiagnosticCode :=
            c_uiDiagnosticResetNotRequired;
    ELSIF NOT xEquipmentStopped THEN
        xResetRejected := TRUE;
        stSafety.uiDiagnosticCode :=
            c_uiDiagnosticEquipmentRunning;
    ELSIF xStandardControlPermitRequest THEN
        xResetRejected := TRUE;
        stSafety.uiDiagnosticCode :=
            c_uiDiagnosticPermitRequestActive;
    ELSE
        xResetRequiredLatched := FALSE;
        xResetAccepted := TRUE;
        stSafety.udiLastAcceptedResetSequence :=
            udiResetSequence;
        stSafety.uiDiagnosticCode := c_uiDiagnosticNone;
    END_IF;
END_IF;

(* State and standard-control permits are derived fail-closed each scan. *)
IF NOT xFeedbackValid THEN
    stSafety.eState := SafetyUnknown;
    stSafety.uiDiagnosticCode :=
        c_uiDiagnosticFeedbackInvalid;
ELSIF xEmergencyActive THEN
    stSafety.eState := SafetyTripActive;
    stSafety.uiDiagnosticCode :=
        c_uiDiagnosticEmergencyActive;
ELSIF NOT xSafetyRelayHealthy THEN
    stSafety.eState := SafetyTripActive;
    stSafety.uiDiagnosticCode :=
        c_uiDiagnosticSafetyRelay;
ELSIF NOT xSTOFeedbackHealthy THEN
    stSafety.eState := SafetyFeedbackFault;
    stSafety.uiDiagnosticCode :=
        c_uiDiagnosticSTOFeedback;
ELSIF NOT xContactorFeedbackHealthy THEN
    stSafety.eState := SafetyFeedbackFault;
    stSafety.uiDiagnosticCode :=
        c_uiDiagnosticContactorFeedback;
ELSIF xResetRequiredLatched THEN
    stSafety.eState := SafetyResetRequired;
    IF NOT xResetRejected THEN
        stSafety.uiDiagnosticCode := c_uiDiagnosticNone;
    END_IF;
ELSIF xStandardControlPermitRequest AND
      NOT xResetAccepted THEN
    stSafety.eState := SafetyHealthyPermitted;
    IF NOT xResetRejected THEN
        stSafety.uiDiagnosticCode := c_uiDiagnosticNone;
    END_IF;
    stSafety.xAutomaticPermitted := TRUE;
    stSafety.xMotionPermitted := TRUE;
    stSafety.xBlowerPermitted := TRUE;
    stSafety.xDosingPermitted := TRUE;
ELSE
    stSafety.eState := SafetyHealthyStopped;
    IF NOT xResetRejected THEN
        stSafety.uiDiagnosticCode := c_uiDiagnosticNone;
    END_IF;
END_IF;

stSafety.xRecoveryPermitted :=
    xAllObservedHealthy AND
    NOT xResetRequiredLatched AND
    NOT xResetAccepted AND
    xEquipmentStopped;

stSafety.xFeedbackValid := xFeedbackValid;
stSafety.xEmergencyActive := xEmergencyActive;
stSafety.xSafetyRelayHealthy := xSafetyRelayHealthy;
stSafety.xSTOFeedbackHealthy := xSTOFeedbackHealthy;
stSafety.xContactorFeedbackHealthy :=
    xContactorFeedbackHealthy;
stSafety.xResetRequired := xResetRequiredLatched;

END_FUNCTION_BLOCK

(* ---- FB_Selector.st ---- *)
FUNCTION_BLOCK FB_Selector
VAR_INPUT
    xEnable : BOOL;
    xHomeRequest : BOOL;
    xMoveRequest : BOOL;
    uiTargetOutlet : UINT;
    udiCommandSequence : UDINT;
    udiResetSequence : UDINT;
    xStopRequest : BOOL;
    xServicePermission : BOOL;
    xSafetyOK : BOOL;
    diPosition : DINT;
    xPositionValid : BOOL;
    xLeftLimit : BOOL;
    xRightLimit : BOOL;
    xMotorRunning : BOOL;
    xMotorFault : BOOL;
    stConfig : ST_SelectorConfig;
    udiMonotonicTickMs : UDINT;
END_VAR
VAR_OUTPUT
    eState : E_SelectorState := SelectorDisabled;
    xMoveLeftRequest : BOOL;
    xMoveRightRequest : BOOL;
    xReady : BOOL;
    xMoving : BOOL;
    xInPosition : BOOL;
    uiCurrentOutlet : UINT;
    uiDiagnosticCode : UINT;
    udiLastAcceptedSequence : UDINT;
END_VAR
VAR
    uiLatchedTargetOutlet : UINT;
    diLatchedTargetPosition : DINT;
    udiMoveStartTickMs : UDINT;
    udiSettleStartTickMs : UDINT;
    udiLastResetSequence : UDINT;
    xHasAcceptedCommand : BOOL;
    xHasAcceptedReset : BOOL;
    diPositionError : DINT;
    diForwardDistance : DINT;
    diReverseDistance : DINT;
    diDistanceToTarget : DINT;
    iOutlet : INT;
    iTargetOutlet : INT;
    uiPositionMatchCount : UINT;
    xConfigValid : BOOL;
    xTargetValid : BOOL;
    xLogicalLeft : BOOL;
END_VAR
VAR CONSTANT
    c_uiDiagnosticNone : UINT := 0;
    c_uiDiagnosticConfig : UINT := 10;
    c_uiDiagnosticInvalidTarget : UINT := 11;
    c_uiDiagnosticPosition : UINT := 12;
    c_uiDiagnosticMotorFault : UINT := 13;
    c_uiDiagnosticLeftLimit : UINT := 14;
    c_uiDiagnosticRightLimit : UINT := 15;
    c_uiDiagnosticTimeout : UINT := 16;
    c_uiDiagnosticSafety : UINT := 17;
    c_uiDiagnosticStopped : UINT := 18;
    c_uiDiagnosticFeedback : UINT := 19;
END_VAR

xMoveLeftRequest := FALSE;
xMoveRightRequest := FALSE;
xReady := FALSE;
xMoving := FALSE;
xInPosition := FALSE;

xConfigValid := (stConfig.uiOutletCount >= 1) AND
                (stConfig.uiOutletCount <= 64) AND
                (stConfig.diPositionTolerance > 0) AND
                (stConfig.diAnalogMinimum < stConfig.diAnalogMaximum) AND
                (stConfig.udiSettleTimeMs > 0) AND
                (stConfig.udiMoveTimeoutMs > 0) AND
                stConfig.axOutletCalibrated[1];

IF stConfig.eTravelMode = SelectorLinearLimited THEN
    xConfigValid := xConfigValid AND stConfig.xLimitsEnabled;
ELSIF stConfig.eTravelMode = SelectorCyclic360 THEN
    xConfigValid := xConfigValid AND
                    stConfig.xAbsolutePositionFeedback AND
                    (stConfig.diCycleLength > (2 * stConfig.diPositionTolerance)) AND
                    (stConfig.diAnalogMinimum = 0) AND
                    (stConfig.diAnalogMaximum = (stConfig.diCycleLength - 1));
ELSE
    xConfigValid := FALSE;
END_IF;

IF NOT xEnable THEN
    eState := SelectorDisabled;
    uiCurrentOutlet := 0;
    uiDiagnosticCode := c_uiDiagnosticNone;
ELSIF NOT xSafetyOK THEN
    eState := SelectorFault;
    uiCurrentOutlet := 0;
    uiDiagnosticCode := c_uiDiagnosticSafety;
ELSIF (stConfig.eTravelMode = SelectorLinearLimited) AND
      stConfig.xLimitsEnabled AND xLeftLimit AND xRightLimit THEN
    eState := SelectorFault;
    uiCurrentOutlet := 0;
    uiDiagnosticCode := c_uiDiagnosticFeedback;
ELSIF xMotorFault THEN
    eState := SelectorFault;
    uiCurrentOutlet := 0;
    uiDiagnosticCode := c_uiDiagnosticMotorFault;
ELSIF NOT xConfigValid THEN
    eState := SelectorFault;
    uiCurrentOutlet := 0;
    uiDiagnosticCode := c_uiDiagnosticConfig;
ELSIF xStopRequest AND (eState <> SelectorFault) THEN
    eState := SelectorInitializing;
    uiCurrentOutlet := 0;
    uiDiagnosticCode := c_uiDiagnosticStopped;
ELSE
    CASE eState OF
        SelectorDisabled:
            eState := SelectorInitializing;
            uiDiagnosticCode := c_uiDiagnosticNone;

        SelectorInitializing:
            uiCurrentOutlet := 0;

            IF NOT xPositionValid OR
               (diPosition < stConfig.diAnalogMinimum) OR
               (diPosition > stConfig.diAnalogMaximum) THEN
                uiDiagnosticCode := c_uiDiagnosticPosition;
            ELSE
                uiPositionMatchCount := 0;

                FOR iOutlet := 1 TO 64 DO
                    IF (iOutlet <= UINT_TO_INT(stConfig.uiOutletCount)) AND
                       stConfig.axOutletCalibrated[iOutlet] AND
                       (((stConfig.eTravelMode = SelectorLinearLimited) AND
                         (ABS(diPosition -
                              stConfig.adiOutletPosition[iOutlet]) <=
                          stConfig.diPositionTolerance)) OR
                        ((stConfig.eTravelMode = SelectorCyclic360) AND
                         (F_CyclicDistance(
                              diCurrentPosition := diPosition,
                              diTargetPosition :=
                                  stConfig.adiOutletPosition[iOutlet],
                              diCycleLength := stConfig.diCycleLength) <=
                          stConfig.diPositionTolerance))) THEN
                        uiCurrentOutlet := INT_TO_UINT(iOutlet);
                        uiPositionMatchCount := uiPositionMatchCount + 1;
                    END_IF;
                END_FOR;

                IF uiPositionMatchCount > 1 THEN
                    uiCurrentOutlet := 0;
                    eState := SelectorFault;
                    uiDiagnosticCode := c_uiDiagnosticConfig;
                ELSIF uiCurrentOutlet > 0 THEN
                    eState := SelectorReady;
                    uiDiagnosticCode := c_uiDiagnosticNone;
                ELSIF xHomeRequest AND
                      (NOT xHasAcceptedCommand OR
                       (udiCommandSequence <> udiLastAcceptedSequence)) THEN
                    udiLastAcceptedSequence := udiCommandSequence;
                    xHasAcceptedCommand := TRUE;
                    udiMoveStartTickMs := udiMonotonicTickMs;
                    eState := SelectorHoming;
                    uiDiagnosticCode := c_uiDiagnosticNone;
                END_IF;
            END_IF;

        SelectorHoming:
            xMoving := TRUE;

            IF NOT xPositionValid THEN
                eState := SelectorFault;
                uiDiagnosticCode := c_uiDiagnosticPosition;
            ELSIF stConfig.eTravelMode = SelectorCyclic360 THEN
                diLatchedTargetPosition := stConfig.adiOutletPosition[1];
                uiLatchedTargetOutlet := 1;
                udiMoveStartTickMs := udiMonotonicTickMs;
                eState := SelectorMoving;
            ELSIF xLeftLimit THEN
                diLatchedTargetPosition := stConfig.adiOutletPosition[1];
                uiLatchedTargetOutlet := 1;
                udiSettleStartTickMs := udiMonotonicTickMs;
                eState := SelectorSettling;
            ELSIF F_ElapsedMs(udiCurrentTickMs := udiMonotonicTickMs,
                             udiStartTickMs := udiMoveStartTickMs) >=
                  stConfig.udiMoveTimeoutMs THEN
                eState := SelectorFault;
                uiDiagnosticCode := c_uiDiagnosticTimeout;
            ELSE
                xMoveLeftRequest := NOT stConfig.xReverseDirection;
                xMoveRightRequest := stConfig.xReverseDirection;
            END_IF;

        SelectorReady:
            xReady := TRUE;
            xInPosition := TRUE;

            IF xMotorRunning THEN
                eState := SelectorFault;
                uiDiagnosticCode := c_uiDiagnosticFeedback;
            ELSIF xMoveRequest AND
                  (NOT xHasAcceptedCommand OR
                   (udiCommandSequence <> udiLastAcceptedSequence)) THEN
                udiLastAcceptedSequence := udiCommandSequence;
                xHasAcceptedCommand := TRUE;
                xReady := FALSE;
                xInPosition := FALSE;
                xTargetValid := (uiTargetOutlet >= 1) AND
                                (uiTargetOutlet <= stConfig.uiOutletCount);

                IF xTargetValid THEN
                    iTargetOutlet := UINT_TO_INT(uiTargetOutlet);
                    xTargetValid :=
                        stConfig.axOutletCalibrated[iTargetOutlet] AND
                        (stConfig.adiOutletPosition[iTargetOutlet] >=
                         stConfig.diAnalogMinimum) AND
                        (stConfig.adiOutletPosition[iTargetOutlet] <=
                         stConfig.diAnalogMaximum);
                END_IF;

                IF NOT xTargetValid THEN
                    uiDiagnosticCode := c_uiDiagnosticInvalidTarget;
                ELSE
                    uiLatchedTargetOutlet := uiTargetOutlet;
                    diLatchedTargetPosition :=
                        stConfig.adiOutletPosition[iTargetOutlet];
                    uiCurrentOutlet := 0;
                    udiMoveStartTickMs := udiMonotonicTickMs;
                    eState := SelectorMoving;
                    uiDiagnosticCode := c_uiDiagnosticNone;
                END_IF;
            END_IF;

        SelectorMoving:
            xMoving := TRUE;

            IF NOT xPositionValid OR
               (diPosition < stConfig.diAnalogMinimum) OR
               (diPosition > stConfig.diAnalogMaximum) THEN
                eState := SelectorFault;
                uiDiagnosticCode := c_uiDiagnosticPosition;
            ELSE
                IF stConfig.eTravelMode = SelectorCyclic360 THEN
                    diDistanceToTarget := F_CyclicDistance(
                        diCurrentPosition := diPosition,
                        diTargetPosition := diLatchedTargetPosition,
                        diCycleLength := stConfig.diCycleLength);

                    diForwardDistance := diLatchedTargetPosition - diPosition;
                    IF diForwardDistance < 0 THEN
                        diForwardDistance := diForwardDistance +
                                             stConfig.diCycleLength;
                    END_IF;

                    diReverseDistance := diPosition - diLatchedTargetPosition;
                    IF diReverseDistance < 0 THEN
                        diReverseDistance := diReverseDistance +
                                             stConfig.diCycleLength;
                    END_IF;

                    xLogicalLeft := diReverseDistance < diForwardDistance;
                ELSE
                    diPositionError := diLatchedTargetPosition - diPosition;
                    diDistanceToTarget := ABS(diPositionError);
                    xLogicalLeft := diPositionError < 0;
                END_IF;

                IF diDistanceToTarget <= stConfig.diPositionTolerance THEN
                    udiSettleStartTickMs := udiMonotonicTickMs;
                    eState := SelectorSettling;
                ELSIF F_ElapsedMs(udiCurrentTickMs := udiMonotonicTickMs,
                                 udiStartTickMs := udiMoveStartTickMs) >=
                      stConfig.udiMoveTimeoutMs THEN
                    eState := SelectorFault;
                    uiDiagnosticCode := c_uiDiagnosticTimeout;
                ELSE
                    IF (stConfig.eTravelMode = SelectorLinearLimited) AND
                       stConfig.xLimitsEnabled AND
                       xLogicalLeft AND xLeftLimit THEN
                        eState := SelectorFault;
                        uiDiagnosticCode := c_uiDiagnosticLeftLimit;
                    ELSIF (stConfig.eTravelMode = SelectorLinearLimited) AND
                          stConfig.xLimitsEnabled AND
                          NOT xLogicalLeft AND xRightLimit THEN
                        eState := SelectorFault;
                        uiDiagnosticCode := c_uiDiagnosticRightLimit;
                    ELSIF xLogicalLeft THEN
                        xMoveLeftRequest := NOT stConfig.xReverseDirection;
                        xMoveRightRequest := stConfig.xReverseDirection;
                    ELSE
                        xMoveLeftRequest := stConfig.xReverseDirection;
                        xMoveRightRequest := NOT stConfig.xReverseDirection;
                    END_IF;
                END_IF;
            END_IF;

        SelectorSettling:
            IF xMotorRunning THEN
                eState := SelectorFault;
                uiDiagnosticCode := c_uiDiagnosticFeedback;
            ELSIF NOT xPositionValid THEN
                eState := SelectorFault;
                uiDiagnosticCode := c_uiDiagnosticPosition;
            ELSIF ((stConfig.eTravelMode = SelectorLinearLimited) AND
                   (ABS(diPosition - diLatchedTargetPosition) >
                    stConfig.diPositionTolerance)) OR
                  ((stConfig.eTravelMode = SelectorCyclic360) AND
                   (F_CyclicDistance(
                        diCurrentPosition := diPosition,
                        diTargetPosition := diLatchedTargetPosition,
                        diCycleLength := stConfig.diCycleLength) >
                    stConfig.diPositionTolerance)) THEN
                udiMoveStartTickMs := udiMonotonicTickMs;
                eState := SelectorMoving;
            ELSIF F_ElapsedMs(udiCurrentTickMs := udiMonotonicTickMs,
                             udiStartTickMs := udiSettleStartTickMs) >=
                  stConfig.udiSettleTimeMs THEN
                uiCurrentOutlet := uiLatchedTargetOutlet;
                eState := SelectorReady;
                uiDiagnosticCode := c_uiDiagnosticNone;
            END_IF;

        SelectorFault:
            IF (NOT xHasAcceptedReset OR
                (udiResetSequence <> udiLastResetSequence)) AND
               xSafetyOK AND
               NOT xMotorFault AND
               NOT xMotorRunning AND
               xPositionValid THEN
                udiLastResetSequence := udiResetSequence;
                xHasAcceptedReset := TRUE;
                eState := SelectorInitializing;
                uiDiagnosticCode := c_uiDiagnosticNone;
            END_IF;

    ELSE
        eState := SelectorFault;
        uiCurrentOutlet := 0;
        uiDiagnosticCode := c_uiDiagnosticConfig;
    END_CASE;
END_IF;

(* Logical outputs are always mutually exclusive. *)
IF xMoveLeftRequest AND xMoveRightRequest THEN
    xMoveLeftRequest := FALSE;
    xMoveRightRequest := FALSE;
    eState := SelectorFault;
    uiDiagnosticCode := c_uiDiagnosticFeedback;
END_IF;

END_FUNCTION_BLOCK

(* ---- FB_SystemManager.st ---- *)
FUNCTION_BLOCK FB_SystemManager
VAR_INPUT
    xEnable : BOOL;
    xStart : BOOL;
    xStop : BOOL;
    xPause : BOOL;
    xReset : BOOL;

    xAutoRequest : BOOL;
    xManualRequest : BOOL;
    xServiceRequest : BOOL;
    xSimulationRequest : BOOL;

    xEmergencyStop : BOOL;
    xSafetyOK : BOOL;
    xBlockingFault : BOOL;
    xAllRequiredLinesReady : BOOL;
    xAnyLineRunning : BOOL;
    xAllLinesStopped : BOOL;
    xDesktopCommunicationOK : BOOL;
    xAlarmActive : BOOL;

    xFeedingActive : BOOL;
    usiCurrentLine : USINT;
    uiActiveRecipeId : UINT;
    udiCurrentJobId : UDINT;
END_VAR
VAR_IN_OUT
    stSystemStatus : ST_SystemStatus;
END_VAR
VAR_OUTPUT
    xSystemReady : BOOL;
    xLineEnable : BOOL;
    xModeConflict : BOOL;
    xResetAccepted : BOOL;
END_VAR
VAR
    eState : E_SystemState := SYSTEM_OFF;
    uiRequestedModeCount : UINT;
    xAutoModeValid : BOOL;
    xStartEdge : BOOL;
    xStopEdge : BOOL;
    xPauseEdge : BOOL;
    xResetEdge : BOOL;
    xPreviousStart : BOOL;
    xPreviousStop : BOOL;
    xPreviousPause : BOOL;
    xPreviousReset : BOOL;
END_VAR

xStartEdge := xStart AND NOT xPreviousStart;
xStopEdge := xStop AND NOT xPreviousStop;
xPauseEdge := xPause AND NOT xPreviousPause;
xResetEdge := xReset AND NOT xPreviousReset;
xResetAccepted := FALSE;

uiRequestedModeCount := 0;
IF xAutoRequest THEN
    uiRequestedModeCount := uiRequestedModeCount + 1;
END_IF;
IF xManualRequest THEN
    uiRequestedModeCount := uiRequestedModeCount + 1;
END_IF;
IF xServiceRequest THEN
    uiRequestedModeCount := uiRequestedModeCount + 1;
END_IF;
IF xSimulationRequest THEN
    uiRequestedModeCount := uiRequestedModeCount + 1;
END_IF;

xModeConflict := uiRequestedModeCount > 1;
xAutoModeValid := xAutoRequest AND
                  (uiRequestedModeCount = 1);

IF xEmergencyStop THEN
    eState := SYSTEM_EMERGENCY;
ELSIF NOT xSafetyOK OR xBlockingFault THEN
    eState := SYSTEM_FAULT;
ELSIF NOT xEnable THEN
    eState := SYSTEM_OFF;
ELSE
    CASE eState OF
        SYSTEM_OFF:
            eState := SYSTEM_INITIALIZING;

        SYSTEM_INITIALIZING:
            IF (uiRequestedModeCount = 1) AND
               xAllRequiredLinesReady THEN
                eState := SYSTEM_READY;
            END_IF;

        SYSTEM_READY:
            IF xStopEdge THEN
                eState := SYSTEM_STOPPING;
            ELSIF (uiRequestedModeCount <> 1) THEN
                eState := SYSTEM_INITIALIZING;
            ELSIF xStartEdge AND xAutoModeValid AND
                  xAllRequiredLinesReady THEN
                eState := SYSTEM_RUNNING;
            END_IF;

        SYSTEM_RUNNING:
            IF xStopEdge OR NOT xAutoModeValid THEN
                eState := SYSTEM_STOPPING;
            ELSIF xPauseEdge THEN
                eState := SYSTEM_PAUSED;
            END_IF;

        SYSTEM_PAUSED:
            IF xStopEdge OR NOT xAutoModeValid THEN
                eState := SYSTEM_STOPPING;
            ELSIF xStartEdge AND
                  xAllRequiredLinesReady THEN
                eState := SYSTEM_RUNNING;
            END_IF;

        SYSTEM_STOPPING:
            IF xAllLinesStopped THEN
                IF (uiRequestedModeCount = 1) AND
                   xAllRequiredLinesReady THEN
                    eState := SYSTEM_READY;
                ELSE
                    eState := SYSTEM_INITIALIZING;
                END_IF;
            END_IF;

        SYSTEM_FAULT:
            IF xResetEdge AND xAllLinesStopped THEN
                xResetAccepted := TRUE;
                eState := SYSTEM_INITIALIZING;
            END_IF;

        SYSTEM_EMERGENCY:
            IF xResetEdge AND xAllLinesStopped THEN
                xResetAccepted := TRUE;
                eState := SYSTEM_INITIALIZING;
            END_IF;

    ELSE
        eState := SYSTEM_FAULT;
    END_CASE;
END_IF;

xSystemReady := eState = SYSTEM_READY;
xLineEnable := xAutoModeValid AND
               xSafetyOK AND
               NOT xEmergencyStop AND
               NOT xBlockingFault AND
               ((eState = SYSTEM_READY) OR
                (eState = SYSTEM_RUNNING) OR
                (eState = SYSTEM_PAUSED));

stSystemStatus.SystemState := eState;
stSystemStatus.SystemReady := xSystemReady;
stSystemStatus.SystemRunning := eState = SYSTEM_RUNNING;
stSystemStatus.SystemPaused := eState = SYSTEM_PAUSED;
stSystemStatus.SystemStopped := xAllLinesStopped AND
                                NOT xAnyLineRunning AND
                                (eState <> SYSTEM_RUNNING) AND
                                (eState <> SYSTEM_PAUSED) AND
                                (eState <> SYSTEM_STOPPING);
stSystemStatus.AutoMode := xAutoModeValid;
stSystemStatus.ManualMode := xManualRequest AND
                             (uiRequestedModeCount = 1);
stSystemStatus.ServiceMode := xServiceRequest AND
                              (uiRequestedModeCount = 1);
stSystemStatus.SimulationMode :=
    xSimulationRequest AND (uiRequestedModeCount = 1);
stSystemStatus.ModeConflict := xModeConflict;
stSystemStatus.SafetyOK := xSafetyOK;
stSystemStatus.EmergencyStop := xEmergencyStop;
stSystemStatus.BlockingFault := xBlockingFault;
stSystemStatus.AlarmActive := xAlarmActive;
stSystemStatus.DesktopCommunicationOK :=
    xDesktopCommunicationOK;
stSystemStatus.AllRequiredLinesReady :=
    xAllRequiredLinesReady;
stSystemStatus.AnyLineRunning := xAnyLineRunning;
stSystemStatus.FeedingActive :=
    xFeedingActive AND xAnyLineRunning;

IF stSystemStatus.FeedingActive THEN
    stSystemStatus.CurrentLine := usiCurrentLine;
    stSystemStatus.ActiveRecipeId := uiActiveRecipeId;
    stSystemStatus.CurrentJobId := udiCurrentJobId;
ELSE
    stSystemStatus.CurrentLine := 0;
    stSystemStatus.ActiveRecipeId := 0;
    stSystemStatus.CurrentJobId := 0;
END_IF;

xPreviousStart := xStart;
xPreviousStop := xStop;
xPreviousPause := xPause;
xPreviousReset := xReset;

END_FUNCTION_BLOCK

(* ---- FB_TimeService.st ---- *)
FUNCTION_BLOCK FB_TimeService
VAR_INPUT
    udiRuntimeTickMs : UDINT;
    xRuntimeTickHealthy : BOOL;
    dtObservedUtc : DT;
    udiSyncSequence : UDINT;
    xSyncRequest : BOOL;
END_VAR
VAR_OUTPUT
    stTime : ST_TimeService;
    xSyncAccepted : BOOL;
    xSyncRejected : BOOL;
    uiResultCode : UINT;
END_VAR
VAR
    xInitialized : BOOL;
    xPreviousSyncRequest : BOOL;
    xHasAcceptedSync : BOOL;
    udiPreviousRuntimeTickMs : UDINT;
    udiAccumulatedMs : UDINT;
    udiDeltaMs : UDINT;
    udiElapsedSeconds : UDINT;
END_VAR
VAR CONSTANT
    c_uiResultNone : UINT := 0;
    c_uiResultSequenceSaturated : UINT := 1;
    c_uiResultSyncReplay : UINT := 10;
    c_uiResultUtcOutOfRange : UINT := 11;
    c_uiDiagnosticMonotonicUnhealthy : UINT := 20;
END_VAR

stTime.xOneSecondTick := FALSE;
xSyncAccepted := FALSE;
xSyncRejected := FALSE;
uiResultCode := c_uiResultNone;

IF NOT xInitialized THEN
    udiPreviousRuntimeTickMs := udiRuntimeTickMs;
    stTime.udiMonotonicTickMs := udiRuntimeTickMs;
    stTime.xMonotonicHealthy := xRuntimeTickHealthy;

    IF NOT xRuntimeTickHealthy THEN
        stTime.uiTimeDiagnosticCode := c_uiDiagnosticMonotonicUnhealthy;
    END_IF;

    xInitialized := TRUE;
ELSE
    IF udiRuntimeTickMs >= udiPreviousRuntimeTickMs THEN
        udiDeltaMs := udiRuntimeTickMs - udiPreviousRuntimeTickMs;
    ELSE
        udiDeltaMs := (c_udiCounterMaximum - udiPreviousRuntimeTickMs) + udiRuntimeTickMs + 1;
    END_IF;

    udiPreviousRuntimeTickMs := udiRuntimeTickMs;
    stTime.udiMonotonicTickMs := udiRuntimeTickMs;
    stTime.xMonotonicHealthy := xRuntimeTickHealthy;

    IF xRuntimeTickHealthy THEN
        IF udiDeltaMs > (c_udiCounterMaximum - udiAccumulatedMs) THEN
            udiAccumulatedMs := c_udiCounterMaximum;
        ELSE
            udiAccumulatedMs := udiAccumulatedMs + udiDeltaMs;
        END_IF;

        udiElapsedSeconds := udiAccumulatedMs / 1000;

        IF udiElapsedSeconds > 0 THEN
            udiAccumulatedMs := udiAccumulatedMs MOD 1000;
            stTime.xOneSecondTick := TRUE;

            IF udiElapsedSeconds > (c_udiCounterMaximum - stTime.udiMonotonicSecondSequence) THEN
                stTime.udiMonotonicSecondSequence := c_udiCounterMaximum;
                stTime.uiTimeDiagnosticCode := c_uiResultSequenceSaturated;
                uiResultCode := c_uiResultSequenceSaturated;
            ELSE
                stTime.udiMonotonicSecondSequence := stTime.udiMonotonicSecondSequence + udiElapsedSeconds;
                stTime.uiTimeDiagnosticCode := c_uiResultNone;
            END_IF;
        ELSE
            stTime.uiTimeDiagnosticCode := c_uiResultNone;
        END_IF;
    ELSE
        udiAccumulatedMs := 0;
        stTime.uiTimeDiagnosticCode := c_uiDiagnosticMonotonicUnhealthy;
    END_IF;
END_IF;

IF xSyncRequest AND NOT xPreviousSyncRequest THEN
    IF xHasAcceptedSync AND (udiSyncSequence = stTime.udiLastAcceptedSyncSequence) THEN
        xSyncRejected := TRUE;
        uiResultCode := c_uiResultSyncReplay;
    ELSIF (dtObservedUtc < DT#2020-01-01-00:00:00) OR
          (dtObservedUtc > DT#2100-12-31-23:59:59) THEN
        xSyncRejected := TRUE;
        uiResultCode := c_uiResultUtcOutOfRange;
    ELSE
        stTime.dtObservedUtc := dtObservedUtc;
        stTime.udiLastAcceptedSyncSequence := udiSyncSequence;
        stTime.xWallClockValid := TRUE;
        xHasAcceptedSync := TRUE;
        xSyncAccepted := TRUE;
    END_IF;
END_IF;

xPreviousSyncRequest := xSyncRequest;

END_FUNCTION_BLOCK
